% RSLogix 500 project 7.6.RSS, saved by version 8.30.00.16 %
PROJECT "7.6"    % processor: Bul.1763 MicroLogix 1100 Series B %

PROGRAM FILES
  LAD 2   4 rungs

DATA FILES
  O0 OUTPUT  4 elements
  I1 INPUT  6 elements
  S2 STATUS  66 elements
  B3 BINARY  1 elements
  T4 TIMER  2 elements
  C5 COUNTER  1 elements
  R6 CONTROL  1 elements
  N7 INTEGER  1 elements
  F8 FLOAT  1 elements

LADDER 2
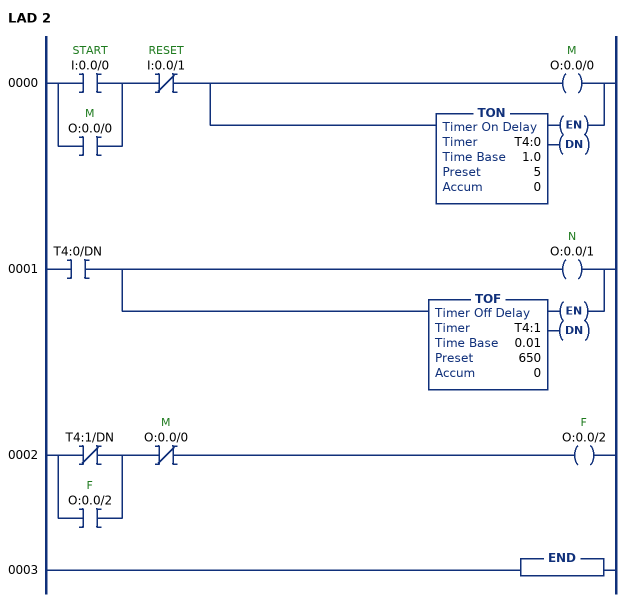
% Rung: 0 %
SOR BST XIC I:0.0/0 NXB XIC O:0.0/0 BND XIO I:0.0/1 BST OTE O:0.0/0 NXB TON T4:0 1.0 5 0 BND EOR
%   I:0.0/0  "START" %
%   O:0.0/0  "M" %
%   I:0.0/1  "RESET" %
% Rung: 1 %
SOR XIC T4:0/DN BST OTE O:0.0/1 NXB TOF T4:1 0.01 650 0 BND EOR
%   O:0.0/1  "N" %
% Rung: 2 %
SOR BST XIO T4:1/DN NXB XIC O:0.0/2 BND XIO O:0.0/0 OTE O:0.0/2 EOR
%   O:0.0/2  "F" %
%   O:0.0/0  "M" %
% Rung: 3 %
SOR END EOR

DATA TABLE (non-zero values as saved)
DATA T4
% .PRE .ACC %
% T4:0 % 5 0
% T4:1 % 650 0
